SUBAPPLICATION Uebung_020c_AX (* DigitalInput_I1 auf DigitalOutput_Q1; E_TON; Einschaltverzögert *)
  (* Standard: 61499-2; Description: Copyright (c) 2023 Meisterschulen am Ostbahnhof This program and the accompanying materials are made available under the terms of the Eclipse Public License 2.0 which is available at https://www.eclipse.org/legal/epl-2.0/ SPDX-License-Identifier: EPL-2.0 *)
  (* Version 1.0, 2023-10-23, Franz Höpfinger, Meisterschulen am Ostbahnhof *)
  PACKAGE Uebungen;
  IMPORT logiBUS::io::DI::logiBUS_DI::Input_I1;
  IMPORT logiBUS::io::DQ::logiBUS_DO::Output_Q1;
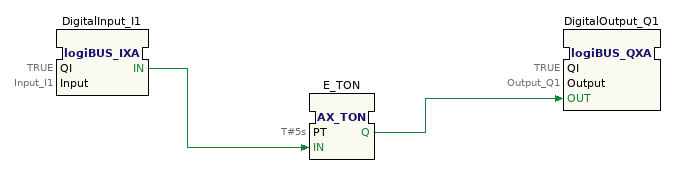
  FBS
    DigitalOutput_Q1 : logiBUS::io::DQ::logiBUS_QXA(QI := TRUE, Output := Output_Q1);
    DigitalInput_I1 : logiBUS::io::DI::logiBUS_IXA(QI := TRUE, Input := Input_I1);
    E_TON : adapter::events::unidirectional::timers::AX_TON(PT := T#5s);
  END_FBS
  ADAPTER_CONNECTIONS
    E_TON.Q TO DigitalOutput_Q1.OUT;
    DigitalInput_I1.IN TO E_TON.IN;
  END_CONNECTIONS
END_SUBAPPLICATION
